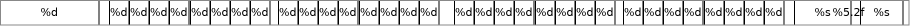
VISUALIZATION visuDataDisplay  // 910x26
VAR_IN_OUT
	d:dutDWord; //data for faceplate
END_VAR
    Rectangle (0,0 99x25), "%d", text variable: d.memLoc
    Rectangle (109,0 20x25), "%d", text variable: d.b38, colour toggle: d.b38
    Rectangle (129,0 20x25), "%d", text variable: d.b37, colour toggle: d.b37
    Rectangle (149,0 20x25), "%d", text variable: d.b36, colour toggle: d.b36
    Rectangle (169,0 20x25), "%d", text variable: d.b35, colour toggle: d.b35
    Rectangle (190,0 20x25), "%d", text variable: d.b34, colour toggle: d.b34
    Rectangle (210,0 20x25), "%d", text variable: d.b33, colour toggle: d.b33
    Rectangle (230,0 20x25), "%d", text variable: d.b32, colour toggle: d.b32
    Rectangle (250,0 20x25), "%d", text variable: d.b31, colour toggle: d.b31
    Rectangle (278,0 20x25), "%d", text variable: d.b28, colour toggle: d.b28
    Rectangle (298,0 20x25), "%d", text variable: d.b27, colour toggle: d.b27
    Rectangle (318,0 20x25), "%d", text variable: d.b26, colour toggle: d.b26
    Rectangle (338,0 20x25), "%d", text variable: d.b25, colour toggle: d.b25
    Rectangle (359,0 20x25), "%d", text variable: d.b24, colour toggle: d.b24
    Rectangle (379,0 20x25), "%d", text variable: d.b23, colour toggle: d.b23
    Rectangle (399,0 20x25), "%d", text variable: d.b22, colour toggle: d.b22
    Rectangle (419,0 20x25), "%d", text variable: d.b21, colour toggle: d.b21
    Rectangle (454,0 20x25), "%d", text variable: d.b18, colour toggle: d.b18
    Rectangle (474,0 20x25), "%d", text variable: d.b17, colour toggle: d.b17
    Rectangle (494,0 20x25), "%d", text variable: d.b16, colour toggle: d.b16
    Rectangle (514,0 20x25), "%d", text variable: d.b15, colour toggle: d.b15
    Rectangle (535,0 20x25), "%d", text variable: d.b14, colour toggle: d.b14
    Rectangle (555,0 20x25), "%d", text variable: d.b13, colour toggle: d.b13
    Rectangle (575,0 20x25), "%d", text variable: d.b12, colour toggle: d.b12
    Rectangle (595,0 20x25), "%d", text variable: d.b11, colour toggle: d.b11
    Rectangle (623,0 20x25), "%d", text variable: d.b08, colour toggle: d.b08
    Rectangle (643,0 20x25), "%d", text variable: d.b07, colour toggle: d.b07
    Rectangle (663,0 20x25), "%d", text variable: d.b06, colour toggle: d.b06
    Rectangle (683,0 20x25), "%d", text variable: d.b05, colour toggle: d.b05
    Rectangle (704,0 20x25), "%d", text variable: d.b04, colour toggle: d.b04
    Rectangle (724,0 20x25), "%d", text variable: d.b03, colour toggle: d.b03
    Rectangle (744,0 20x25), "%d", text variable: d.b02, colour toggle: d.b02
    Rectangle (764,0 20x25), "%d", text variable: d.b01, colour toggle: d.b01
    Rectangle (794,0 57x25), "%s", text variable: d.hexVal, invisible if: d.ShowREAL
    Rectangle (860,0 43x25), "%s", text variable: d.valStr, invisible if: d.ShowREAL
    Rectangle (794,0 109x25), "%5.2f", text variable: d.floatVal, invisible if: d.ShowHex
END_VISUALIZATION

(* stored: Version 1.1.0.1, ProductVersion 3.1.4024.12
   Visu visuDataDisplay: Id {ab253d7b-3a9a-4101-9be3-e8a0fceb6741} *)
